% RSLogix 500 project VFD DRIVE LOGIC.RSS, saved by version 8.30.00.16 %
PROJECT "SIM_PLC"    % processor: Bul.1763 MicroLogix 1100 Series B %

PROGRAM FILES
  LAD 2 "MAIN"  3 rungs
  LAD 3 "IO"  3 rungs
  LAD 4 "CTRL LOGIC"  10 rungs

DATA FILES
  O0 OUTPUT  4 elements
  I1 INPUT  6 elements
  S2 STATUS  66 elements
  B3 BINARY  1 elements
  T4 TIMER  1 elements
  C5 COUNTER  1 elements
  R6 CONTROL  1 elements
  N7 INTEGER  7 elements
  F8 FLOAT  2 elements

LADDER 2 "MAIN"
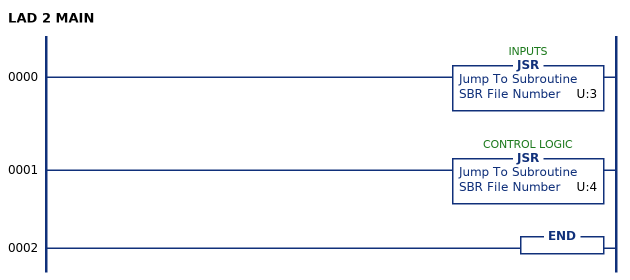
% Rung: 0 %
SOR JSR U:3 EOR
%   U:3  "INPUTS" %
% Rung: 1 %
SOR JSR U:4 EOR
%   U:4  "CONTROL LOGIC" %
% Rung: 2 %
SOR END EOR

LADDER 3 "IO"
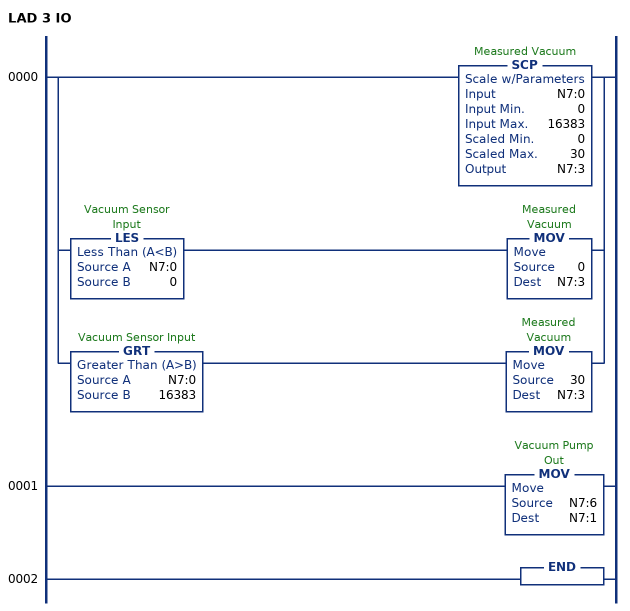
% Rung: 0 %
SOR BST SCP N7:0 0 16383 0 30 N7:3 NXB LES N7:0 0 MOV 0 N7:3 NXB GRT N7:0 16383 MOV 30 N7:3 BND EOR
%   N7:0  "Vacuum Sensor Input" %
%   N7:3  "Measured Vacuum" %
% Rung: 1 %
SOR MOV N7:6 N7:1 EOR
%   N7:6  "Adjusted Vacuum Out" %
%   N7:1  "Vacuum Pump Out" %
% Rung: 2 %
SOR END EOR

LADDER 4 "CTRL LOGIC"
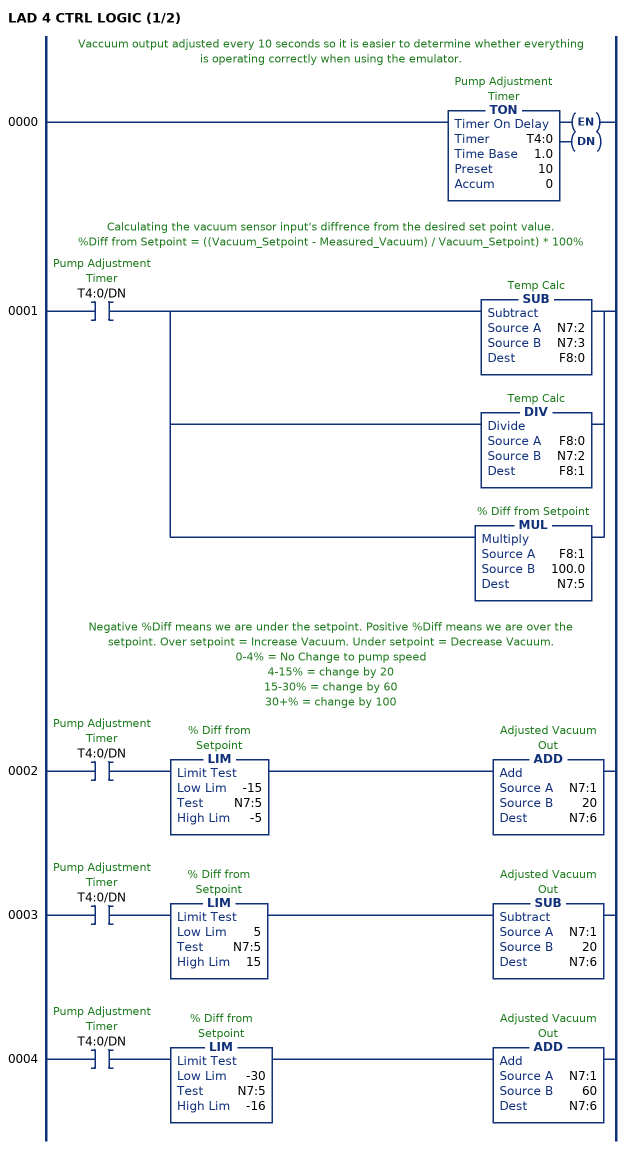
% Rung: 0 %
% Vaccuum output adjusted every 10 seconds so it is easier to determine whether everything is operating correctly when using the emulator. %
SOR TON T4:0 1.0 10 0 EOR
%   T4:0  "Pump Adjustment Timer" %
% Rung: 1 %
% Calculating the vacuum sensor input's diffrence from the desired set point value.
% 
% %Diff from Setpoint = ((Vacuum_Setpoint - Measured_Vacuum) / Vacuum_Setpoint) * 100% %
SOR XIC T4:0/DN BST SUB N7:2 N7:3 F8:0 NXB DIV F8:0 N7:2 F8:1 NXB MUL F8:1 100.0 N7:5 BND EOR
%   T4:0  "Pump Adjustment Timer" %
%   N7:2  "Vacuum Setpoint" %
%   N7:3  "Measured Vacuum" %
%   F8:0  "Temp Calc" %
%   F8:1  "Temp Calc" %
%   N7:5  "% Diff from Setpoint" %
% Rung: 2 %
% Negative %Diff means we are under the setpoint. Positive %Diff means we are over the setpoint. Over setpoint = Increase Vacuum. Under setpoint = Decrease Vacuum.
% 
% 0-4% = No Change to pump speed
% 4-15% = change by 20
% 15-30% = change by 60
% 30+% = change by 100 %
SOR XIC T4:0/DN LIM -15 N7:5 -5 ADD N7:1 20 N7:6 EOR
%   T4:0  "Pump Adjustment Timer" %
%   N7:5  "% Diff from Setpoint" %
%   N7:1  "Vacuum Pump Out" %
%   N7:6  "Adjusted Vacuum Out" %
% Rung: 3 %
SOR XIC T4:0/DN LIM 5 N7:5 15 SUB N7:1 20 N7:6 EOR
%   T4:0  "Pump Adjustment Timer" %
%   N7:5  "% Diff from Setpoint" %
%   N7:1  "Vacuum Pump Out" %
%   N7:6  "Adjusted Vacuum Out" %
% Rung: 4 %
SOR XIC T4:0/DN LIM -30 N7:5 -16 ADD N7:1 60 N7:6 EOR
%   T4:0  "Pump Adjustment Timer" %
%   N7:5  "% Diff from Setpoint" %
%   N7:1  "Vacuum Pump Out" %
%   N7:6  "Adjusted Vacuum Out" %

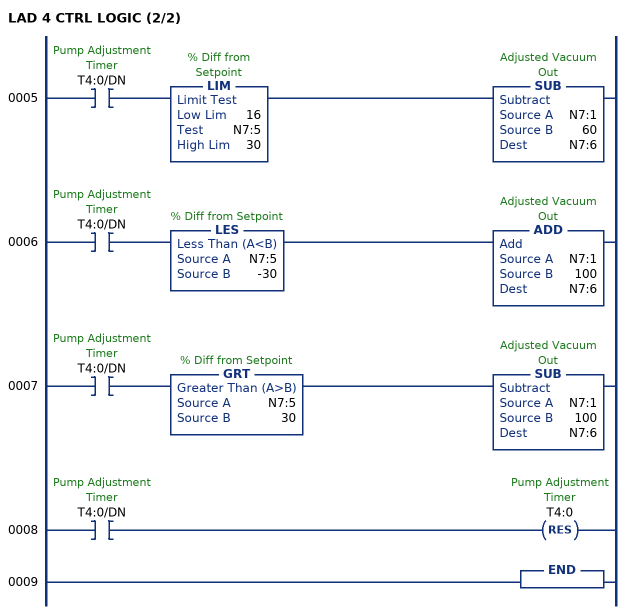
% Rung: 5 %
SOR XIC T4:0/DN LIM 16 N7:5 30 SUB N7:1 60 N7:6 EOR
%   T4:0  "Pump Adjustment Timer" %
%   N7:5  "% Diff from Setpoint" %
%   N7:1  "Vacuum Pump Out" %
%   N7:6  "Adjusted Vacuum Out" %
% Rung: 6 %
SOR XIC T4:0/DN LES N7:5 -30 ADD N7:1 100 N7:6 EOR
%   T4:0  "Pump Adjustment Timer" %
%   N7:5  "% Diff from Setpoint" %
%   N7:1  "Vacuum Pump Out" %
%   N7:6  "Adjusted Vacuum Out" %
% Rung: 7 %
SOR XIC T4:0/DN GRT N7:5 30 SUB N7:1 100 N7:6 EOR
%   T4:0  "Pump Adjustment Timer" %
%   N7:5  "% Diff from Setpoint" %
%   N7:1  "Vacuum Pump Out" %
%   N7:6  "Adjusted Vacuum Out" %
% Rung: 8 %
SOR XIC T4:0/DN RES T4:0 EOR
%   T4:0  "Pump Adjustment Timer" %
% Rung: 9 %
SOR END EOR

OTHER DOCUMENTED ADDRESSES
  N7:4  "Temp Calc"

DATA TABLE (non-zero values as saved)
DATA T4
% .PRE .ACC %
% T4:0 % 10 0
DATA N7
% N7:0 % 8192 0 15 0 0 0 0
